TYPE ST_BaseEvents_RowInQueue :
STRUCT
	uiIDEvent								: UINT;					//unikalny numer zgloszenia dla całego projektu nadawany automatycznie 
	uiIDItem								: UINT;					// unikalny numer elementu w systemie
	bActive									: BOOL;             	
	bIgnoreRepetitions						: BOOL;					//jak true nie zliczaj powtorzeń wystapienia np komunikaty
	uiRepetitionCounter						: UINT;             	
	dtStart									: DT;					//poczatek wystepowania zgłoszenia
	dtFinish								: DT;					//koniec wystepowaniazgloszenia
	dtConfirmed								: DT;					// stempel potwierdzenia 
	bConfirm								: BOOL;					//informacja czy bo byc zgłoszenie potwierdzone
	eEventCategory							: E_BaseEvents_Category;
	eEventAction							: E_BaseEvents_Action;	//okresla rodzaj zgloszenia w kolejce Start stop 
END_STRUCT
END_TYPE

(* stored: Version 1.1.0.1
   DUT ST_BaseEvents_RowInQueue: Id {f444b0ca-18c7-0625-1f7a-9be02a9ec795} *)
